(* IEC 61131-3 sources: stc-rs/lib/src/test/test_decl_parse, 10 files *)

(* ---- test_alias_decl.st ---- *)
TYPE
TestAlias: Int;
END_TYPE

(* ---- test_enum_decl.st ---- *)
TYPE TestEnum:
(
    E1,
    E2 := 10,
    E3
) DINT;
END_TYPE

(* ---- test_struct_declare.st ---- *)
TYPE

MyStruct:
STRUCT
    a: INT;
    b: BOOL;
END_STRUCT

END_TYPE

(* ---- test_base_types.st ---- *)
var_global
    a: BIT;
end_var

(* ---- test_global_var_decl.st ---- *)
var_global
end_var
var_global
a:BYtE;
end_var

(* ---- test_array_decl.st ---- *)
FUNCTION F: INT

VAR
    a: ARRAY [ 1 .. 2 ]  OF INT;
    b:ARRAY[1..2]OF INT;
    c: ARRAY[1.2..2.3]OF DWORD;
    c2: ARRAY[1..3, 2..4]OF DWORD;
    b:ARRAY[a..b]OF INT;
    b2:ARRAY[a..b, c..d]OF INT;
    b3:ARRAY[a..b, c..d]OF ARRAY[0..10] OF INT;
END_VAR

END_FUNCTION

(* ---- test_fun_decl.st ---- *)
function TestFun : INT

VAR RETAIN
    a: INT;
END_VAR

END_FUNCTION

(* ---- test_fun_without_return_type.st ---- *)
Function Test :
VAR
END_VAR
end_function

(* ---- test_parse_prg.st ---- *)
program Task :
end_program

(* ---- test_temp_var.st ---- *)
program Task :
    VAR
        a: BYTE;
    END_VAR

    VAR_TEMP
        b: INT;
    END_VAR
end_program
